// TIA Portal V20 export
FUNCTION "06 T10 LANT Output" : Void   // FC1693, LAD
TITLE = OUTPUT
{ S7_Optimized_Access := 'TRUE' }
// stored: AutoNumber false, SetENOAutomatically false
   VAR_TEMP
      Aux_real : Real;
      Aux_dint : DInt;
      Aux_uint : UInt;
      Aux_Bool : Bool;
      Aux_OS : Bool;
   END_VAR
   VAR_TEMP   // added for the SCL form of the ladder/FBD networks
      _w1 : Bool;
      _w2 : Bool;
      _w3 : Bool;
   END_VAR
BEGIN

REGION Network 1: ============= INTERLOCKS MOVING FORWARD =============
END_REGION

REGION Network 2: Interlocks Move FORWARD - Permanent Conditions
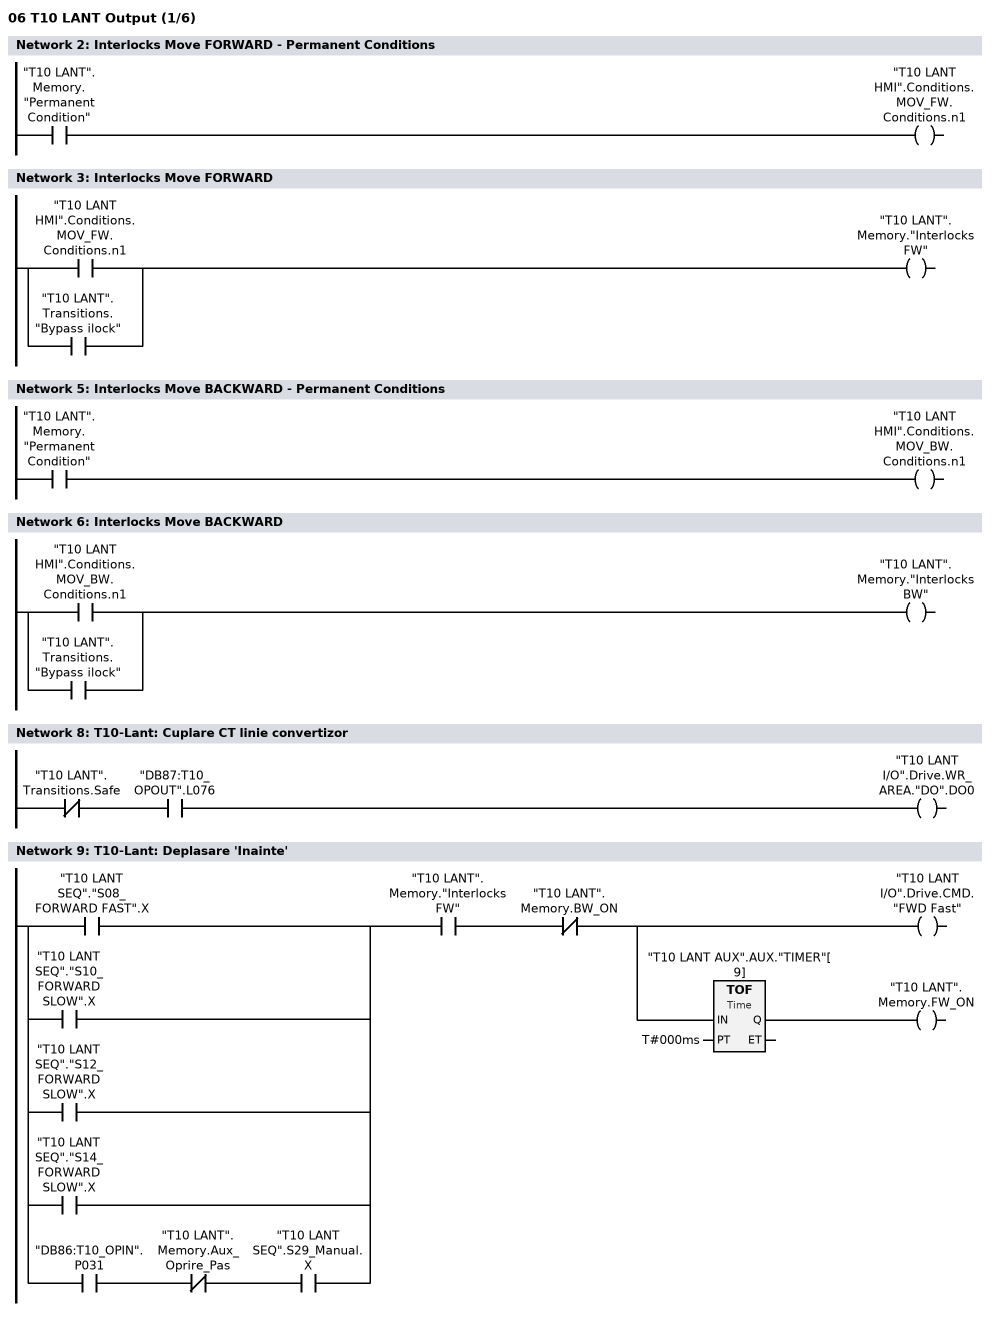
   RUNG wire#powerrail
      Contact( "T10 LANT".Memory."Permanent Condition" )
      Coil( "T10 LANT HMI".Conditions.MOV_FW.Conditions.n1 )
   END_RUNG
   // the same network as SCL:
   "T10 LANT HMI".Conditions.MOV_FW.Conditions.n1 := "T10 LANT".Memory."Permanent Condition";
END_REGION

REGION Network 3: Interlocks Move FORWARD
   RUNG wire#powerrail
      Contact( "T10 LANT HMI".Conditions.MOV_FW.Conditions.n1 )
      wire#w1
      Coil( "T10 LANT".Memory."Interlocks FW" )
   END_RUNG
   RUNG wire#powerrail
      Contact( "T10 LANT".Transitions."Bypass ilock" )
   END_RUNG wire#w1
   // the same network as SCL:
   "T10 LANT".Memory."Interlocks FW" := "T10 LANT HMI".Conditions.MOV_FW.Conditions.n1 OR "T10 LANT".Transitions."Bypass ilock";
END_REGION

REGION Network 4: ============= INTERLOCKS MOVING BACKWARD =============
END_REGION

REGION Network 5: Interlocks Move BACKWARD - Permanent Conditions
   RUNG wire#powerrail
      Contact( "T10 LANT".Memory."Permanent Condition" )
      Coil( "T10 LANT HMI".Conditions.MOV_BW.Conditions.n1 )
   END_RUNG
   // the same network as SCL:
   "T10 LANT HMI".Conditions.MOV_BW.Conditions.n1 := "T10 LANT".Memory."Permanent Condition";
END_REGION

REGION Network 6: Interlocks Move BACKWARD
   RUNG wire#powerrail
      Contact( "T10 LANT HMI".Conditions.MOV_BW.Conditions.n1 )
      wire#w1
      Coil( "T10 LANT".Memory."Interlocks BW" )
   END_RUNG
   RUNG wire#powerrail
      Contact( "T10 LANT".Transitions."Bypass ilock" )
   END_RUNG wire#w1
   // the same network as SCL:
   "T10 LANT".Memory."Interlocks BW" := "T10 LANT HMI".Conditions.MOV_BW.Conditions.n1 OR "T10 LANT".Transitions."Bypass ilock";
END_REGION

REGION Network 7: ============ COMMANDS ============
END_REGION

REGION Network 8: T10-Lant: Cuplare CT linie convertizor
   RUNG wire#powerrail
      I_Contact( "T10 LANT".Transitions.Safe )
      Contact( "DB87:T10_OPOUT".L076 )
      Coil( "T10 LANT I/O".Drive.WR_AREA."DO".DO0 )
   END_RUNG
   // the same network as SCL:
   "T10 LANT I/O".Drive.WR_AREA."DO".DO0 := NOT "T10 LANT".Transitions.Safe AND "DB87:T10_OPOUT".L076;
END_REGION

REGION Network 9: T10-Lant: Deplasare 'Inainte'
   RUNG wire#powerrail
      Contact( "T10 LANT SEQ"."S08_FORWARD FAST".X )
      wire#w1
      Contact( "T10 LANT".Memory."Interlocks FW" )
      I_Contact( "T10 LANT".Memory.BW_ON )
      wire#w2
      Coil( "T10 LANT I/O".Drive.CMD."FWD Fast" )
   END_RUNG
   RUNG wire#powerrail
      Contact( "T10 LANT SEQ"."S10_FORWARD SLOW".X )
   END_RUNG wire#w1
   RUNG wire#powerrail
      Contact( "T10 LANT SEQ"."S12_FORWARD SLOW".X )
   END_RUNG wire#w1
   RUNG wire#powerrail
      Contact( "T10 LANT SEQ"."S14_FORWARD SLOW".X )
   END_RUNG wire#w1
   RUNG wire#powerrail
      Contact( "DB86:T10_OPIN".P031 )
      I_Contact( "T10 LANT".Memory.Aux_Oprire_Pas )
      Contact( "T10 LANT SEQ".S29_Manual.X )
   END_RUNG wire#w1
   RUNG wire#w2
      { S7_Templates := "time_type := Time" } "T10 LANT AUX".AUX."TIMER"[9].TOF(pt := T#000ms, et =>)
      Coil( "T10 LANT".Memory.FW_ON )
   END_RUNG
   // the same network as SCL:
   "T10 LANT I/O".Drive.CMD."FWD Fast" := ("T10 LANT SEQ"."S08_FORWARD FAST".X OR "T10 LANT SEQ"."S10_FORWARD SLOW".X OR "T10 LANT SEQ"."S12_FORWARD SLOW".X OR "T10 LANT SEQ"."S14_FORWARD SLOW".X OR ("DB86:T10_OPIN".P031 AND NOT "T10 LANT".Memory.Aux_Oprire_Pas AND "T10 LANT SEQ".S29_Manual.X)) AND "T10 LANT".Memory."Interlocks FW" AND NOT "T10 LANT".Memory.BW_ON;
   "T10 LANT AUX".AUX."TIMER"[9].TOF(IN := "T10 LANT I/O".Drive.CMD."FWD Fast", PT := T#000ms);
   "T10 LANT".Memory.FW_ON := "T10 LANT AUX".AUX."TIMER"[9].Q;
END_REGION

REGION Network 10: T10-Lant: Deplasare 'Inapoi'
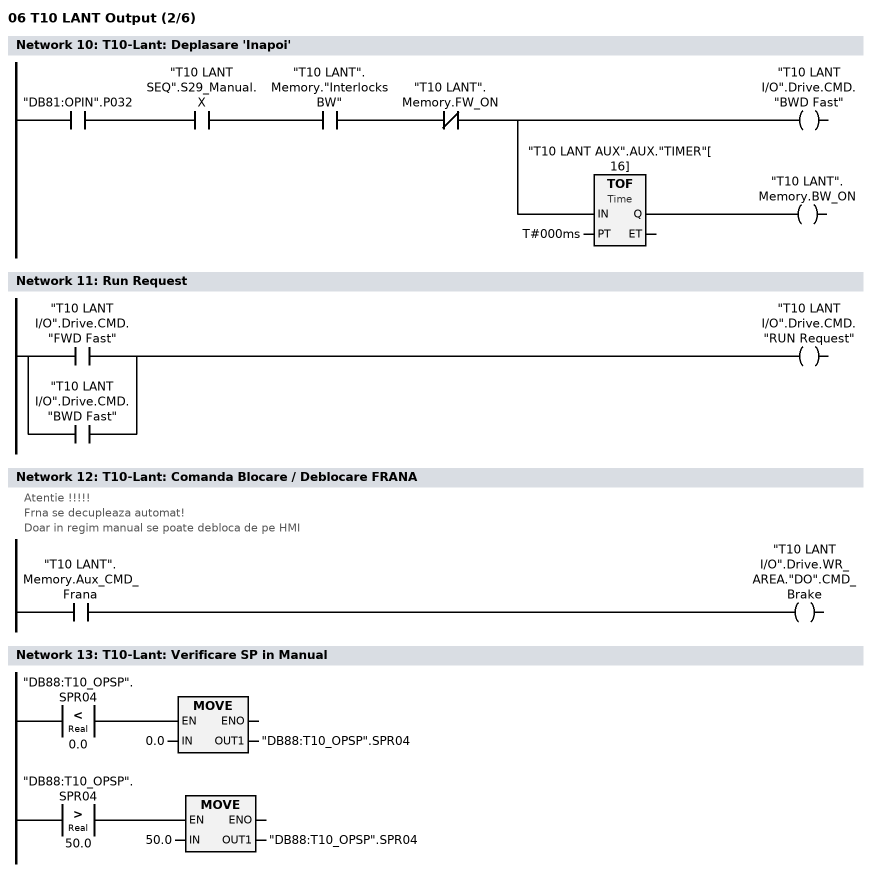
   RUNG wire#powerrail
      Contact( "DB81:OPIN".P032 )
      Contact( "T10 LANT SEQ".S29_Manual.X )
      Contact( "T10 LANT".Memory."Interlocks BW" )
      I_Contact( "T10 LANT".Memory.FW_ON )
      wire#w1
      Coil( "T10 LANT I/O".Drive.CMD."BWD Fast" )
   END_RUNG
   RUNG wire#w1
      { S7_Templates := "time_type := Time" } "T10 LANT AUX".AUX."TIMER"[16].TOF(pt := T#000ms, et =>)
      Coil( "T10 LANT".Memory.BW_ON )
   END_RUNG
   // the same network as SCL:
   "T10 LANT I/O".Drive.CMD."BWD Fast" := "DB81:OPIN".P032 AND "T10 LANT SEQ".S29_Manual.X AND "T10 LANT".Memory."Interlocks BW" AND NOT "T10 LANT".Memory.FW_ON;
   "T10 LANT AUX".AUX."TIMER"[16].TOF(IN := "T10 LANT I/O".Drive.CMD."BWD Fast", PT := T#000ms);
   "T10 LANT".Memory.BW_ON := "T10 LANT AUX".AUX."TIMER"[16].Q;
END_REGION

REGION Network 11: Run Request
   RUNG wire#powerrail
      Contact( "T10 LANT I/O".Drive.CMD."FWD Fast" )
      wire#w1
      Coil( "T10 LANT I/O".Drive.CMD."RUN Request" )
   END_RUNG
   RUNG wire#powerrail
      Contact( "T10 LANT I/O".Drive.CMD."BWD Fast" )
   END_RUNG wire#w1
   // the same network as SCL:
   "T10 LANT I/O".Drive.CMD."RUN Request" := "T10 LANT I/O".Drive.CMD."FWD Fast" OR "T10 LANT I/O".Drive.CMD."BWD Fast";
END_REGION

REGION Network 12: T10-Lant: Comanda Blocare / Deblocare FRANA
   // Atentie !!!!!
   // Frna se decupleaza automat!
   // Doar in regim manual se poate debloca de pe HMI
   RUNG wire#powerrail
      Contact( "T10 LANT".Memory.Aux_CMD_Frana )
      Coil( "T10 LANT I/O".Drive.WR_AREA."DO".CMD_Brake )
   END_RUNG
   // the same network as SCL:
   "T10 LANT I/O".Drive.WR_AREA."DO".CMD_Brake := "T10 LANT".Memory.Aux_CMD_Frana;
END_REGION

REGION Network 13: T10-Lant: Verificare SP in Manual
   RUNG wire#powerrail
      { S7_Templates := "SrcType := Real" } LT_Contact(in1 := "DB88:T10_OPSP".SPR04, in2 := 0.0)
      Move(in := 0.0, out1 => "DB88:T10_OPSP".SPR04)
   END_RUNG
   RUNG wire#powerrail
      { S7_Templates := "SrcType := Real" } GT_Contact(in1 := "DB88:T10_OPSP".SPR04, in2 := 50.0)
      Move(in := 50.0, out1 => "DB88:T10_OPSP".SPR04)
   END_RUNG
   // the same network as SCL:
   IF "DB88:T10_OPSP".SPR04 < 0.0 THEN "DB88:T10_OPSP".SPR04 := 0.0; END_IF;
   IF "DB88:T10_OPSP".SPR04 > 50.0 THEN "DB88:T10_OPSP".SPR04 := 50.0; END_IF;
END_REGION

REGION Network 14: T10-Lant: Ciclu Rapid: Viteza Referinta Incarcare
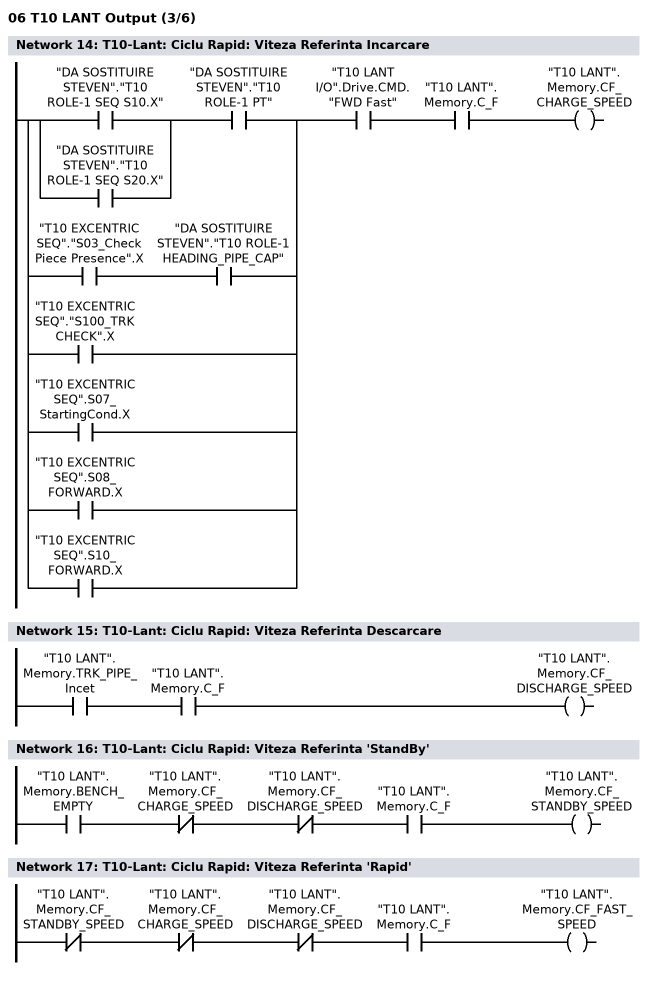
   RUNG wire#powerrail
      Contact( "DA SOSTITUIRE STEVEN"."T10 ROLE-1 SEQ S10.X" )
      wire#w1
      Contact( "DA SOSTITUIRE STEVEN"."T10 ROLE-1 PT" )
      wire#w2
      Contact( "T10 LANT I/O".Drive.CMD."FWD Fast" )
      Contact( "T10 LANT".Memory.C_F )
      Coil( "T10 LANT".Memory.CF_CHARGE_SPEED )
   END_RUNG
   RUNG wire#powerrail
      Contact( "DA SOSTITUIRE STEVEN"."T10 ROLE-1 SEQ S20.X" )
   END_RUNG wire#w1
   RUNG wire#powerrail
      Contact( "T10 EXCENTRIC SEQ"."S03_Check Piece Presence".X )
      Contact( "DA SOSTITUIRE STEVEN"."T10 ROLE-1 HEADING_PIPE_CAP" )
   END_RUNG wire#w2
   RUNG wire#powerrail
      Contact( "T10 EXCENTRIC SEQ"."S100_TRK CHECK".X )
   END_RUNG wire#w2
   RUNG wire#powerrail
      Contact( "T10 EXCENTRIC SEQ".S07_StartingCond.X )
   END_RUNG wire#w2
   RUNG wire#powerrail
      Contact( "T10 EXCENTRIC SEQ".S08_FORWARD.X )
   END_RUNG wire#w2
   RUNG wire#powerrail
      Contact( "T10 EXCENTRIC SEQ".S10_FORWARD.X )
   END_RUNG wire#w2
   // the same network as SCL:
   "T10 LANT".Memory.CF_CHARGE_SPEED := ((("DA SOSTITUIRE STEVEN"."T10 ROLE-1 SEQ S10.X" OR "DA SOSTITUIRE STEVEN"."T10 ROLE-1 SEQ S20.X") AND "DA SOSTITUIRE STEVEN"."T10 ROLE-1 PT") OR ("T10 EXCENTRIC SEQ"."S03_Check Piece Presence".X AND "DA SOSTITUIRE STEVEN"."T10 ROLE-1 HEADING_PIPE_CAP") OR "T10 EXCENTRIC SEQ"."S100_TRK CHECK".X OR "T10 EXCENTRIC SEQ".S07_StartingCond.X OR "T10 EXCENTRIC SEQ".S08_FORWARD.X OR "T10 EXCENTRIC SEQ".S10_FORWARD.X) AND "T10 LANT I/O".Drive.CMD."FWD Fast" AND "T10 LANT".Memory.C_F;
END_REGION

REGION Network 15: T10-Lant: Ciclu Rapid: Viteza Referinta Descarcare
   RUNG wire#powerrail
      Contact( "T10 LANT".Memory.TRK_PIPE_Incet )
      Contact( "T10 LANT".Memory.C_F )
      Coil( "T10 LANT".Memory.CF_DISCHARGE_SPEED )
   END_RUNG
   // the same network as SCL:
   "T10 LANT".Memory.CF_DISCHARGE_SPEED := "T10 LANT".Memory.TRK_PIPE_Incet AND "T10 LANT".Memory.C_F;
END_REGION

REGION Network 16: T10-Lant: Ciclu Rapid: Viteza Referinta 'StandBy'
   RUNG wire#powerrail
      Contact( "T10 LANT".Memory.BENCH_EMPTY )
      I_Contact( "T10 LANT".Memory.CF_CHARGE_SPEED )
      I_Contact( "T10 LANT".Memory.CF_DISCHARGE_SPEED )
      Contact( "T10 LANT".Memory.C_F )
      Coil( "T10 LANT".Memory.CF_STANDBY_SPEED )
   END_RUNG
   // the same network as SCL:
   "T10 LANT".Memory.CF_STANDBY_SPEED := "T10 LANT".Memory.BENCH_EMPTY AND NOT "T10 LANT".Memory.CF_CHARGE_SPEED AND NOT "T10 LANT".Memory.CF_DISCHARGE_SPEED AND "T10 LANT".Memory.C_F;
END_REGION

REGION Network 17: T10-Lant: Ciclu Rapid: Viteza Referinta 'Rapid'
   RUNG wire#powerrail
      I_Contact( "T10 LANT".Memory.CF_STANDBY_SPEED )
      I_Contact( "T10 LANT".Memory.CF_CHARGE_SPEED )
      I_Contact( "T10 LANT".Memory.CF_DISCHARGE_SPEED )
      Contact( "T10 LANT".Memory.C_F )
      Coil( "T10 LANT".Memory.CF_FAST_SPEED )
   END_RUNG
   // the same network as SCL:
   "T10 LANT".Memory.CF_FAST_SPEED := NOT "T10 LANT".Memory.CF_STANDBY_SPEED AND NOT "T10 LANT".Memory.CF_CHARGE_SPEED AND NOT "T10 LANT".Memory.CF_DISCHARGE_SPEED AND "T10 LANT".Memory.C_F;
END_REGION

NETWORK
TITLE = T10-Lant: Viteza Teava 'Inainte' in Mod Automat [%]
// 13.6 m/min ...... 50 Hz
// a m/min...........b Hz
// 
// b=(a*50)/13.6

      A     "T10 LANT".Memory.CF_DISCHARGE_SPEED;
      L     "PRESET POINT ACTIVE".TAB1.P93;  // DISCHARGE SPEE CYCLE
      L     1;
      /I;
      JC    _02;  // ----------------------------
      A     "T10 LANT".Memory.CF_CHARGE_SPEED;
      L     "PRESET POINT ACTIVE".TAB1.P92;  // CHARGE SPEED FAST CYCLE
      L     1;
      /I;
      JC    _02;  // ----------------------------
      A     "T10 LANT".Memory.CF_FAST_SPEED;
      L     "PRESET POINT ACTIVE".TAB1.P90;  // FAST SPEED FAST CYCLE
      L     1;
      /I;
      JC    _02;  // ----------------------------
      A     "T10 LANT".Memory.CF_STANDBY_SPEED;
      L     "PRESET POINT ACTIVE".TAB1.P91;  // STAND-BY SPEED FAST CYCLE
      L     1;
      /I;
      JC    _02;  // ----------------------------
      L     "PRESET POINT ACTIVE".TAB1.P86;  // STANDARD AUTOMATIC CYCLE
      L     1;
      /I;
_02:  NOP   0;  // ----------------------------
      ITD;
      DTR;
      T     "T10 LANT".Memory.SPEED_FW_AUTO_HZ;

      L     "T10 LANT".Memory.SPEED_FW_AUTO_HZ;
      L     50.0;
      *R;
      T     "T10 LANT".Memory.SPEED_FW_AUTO_HZ;

      L     "T10 LANT".Memory.SPEED_FW_AUTO_HZ;
      L     100.0;
      /R;
      T     "T10 LANT".Memory.SPEED_FW_AUTO_HZ;


NETWORK
TITLE = T10-Lant: Viteza Teava 'Inainte' in Mod Manual [%]
// 13.6 m/min ...... 50 Hz
// a m/min...........b Hz
// 
// b=(a*50)/13.6

      L     "PRESET POINT ACTIVE".TAB1.P87;
      L     1;
      /I;
      ITD;
      DTR;
      L     50.0;
      *R;
      L     100.0;
      /R;
      T     #Aux_real;


REGION Network 20: T10-Lant: Comenzi - Setpoint
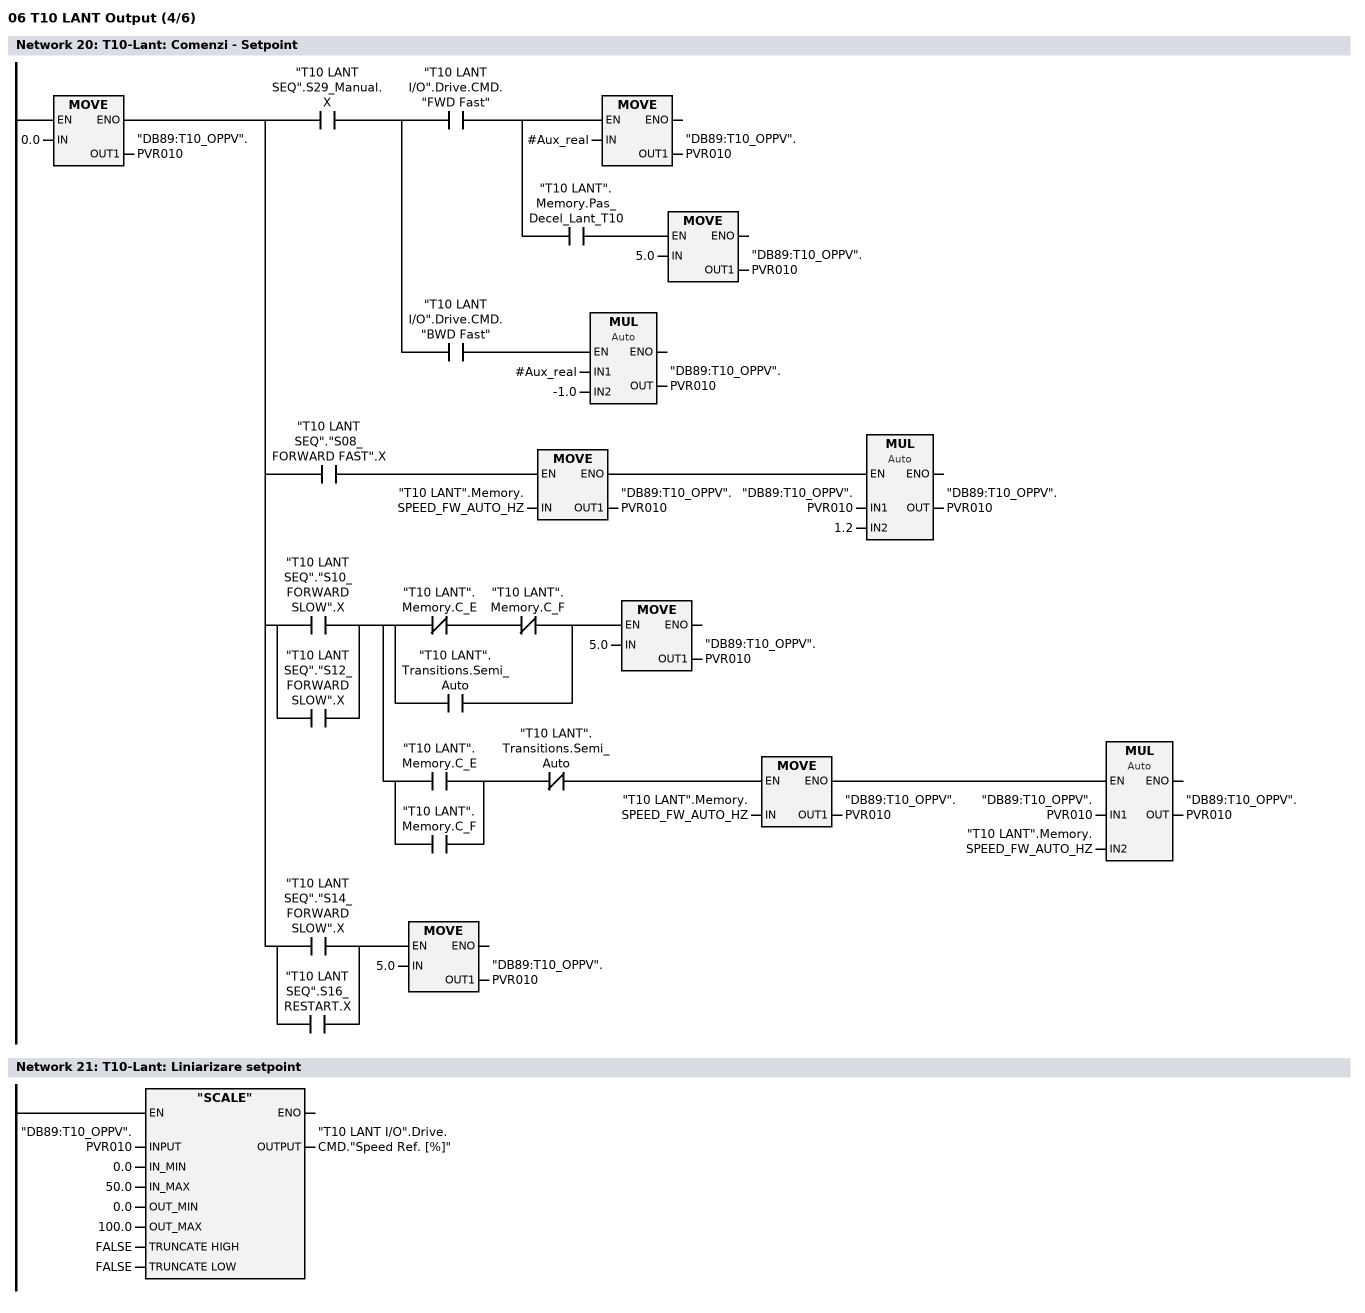
   RUNG wire#powerrail
      Move(in := 0.0, out1 => "DB89:T10_OPPV".PVR010)
      wire#w1
      Contact( "T10 LANT SEQ".S29_Manual.X )
      wire#w2
      Contact( "T10 LANT I/O".Drive.CMD."FWD Fast" )
      wire#w3
      Move(in := #Aux_real, out1 => "DB89:T10_OPPV".PVR010)
   END_RUNG
   RUNG wire#w3
      Contact( "T10 LANT".Memory.Pas_Decel_Lant_T10 )
      Move(in := 5.0, out1 => "DB89:T10_OPPV".PVR010)
   END_RUNG
   RUNG wire#w2
      Contact( "T10 LANT I/O".Drive.CMD."BWD Fast" )
      Mul(in1 := #Aux_real, in2 := -1.0, out => "DB89:T10_OPPV".PVR010)
   END_RUNG
   RUNG wire#w1
      Contact( "T10 LANT SEQ"."S08_FORWARD FAST".X )
      Move(in := "T10 LANT".Memory.SPEED_FW_AUTO_HZ, out1 => "DB89:T10_OPPV".PVR010)
      Mul(in1 := "DB89:T10_OPPV".PVR010, in2 := 1.2, out => "DB89:T10_OPPV".PVR010)
   END_RUNG
   RUNG wire#w1
      Contact( "T10 LANT SEQ"."S10_FORWARD SLOW".X )
      wire#w4
      I_Contact( "T10 LANT".Memory.C_E )
      I_Contact( "T10 LANT".Memory.C_F )
      wire#w5
      Move(in := 5.0, out1 => "DB89:T10_OPPV".PVR010)
   END_RUNG
   RUNG wire#w1
      Contact( "T10 LANT SEQ"."S12_FORWARD SLOW".X )
   END_RUNG wire#w4
   RUNG wire#w4
      Contact( "T10 LANT".Transitions.Semi_Auto )
   END_RUNG wire#w5
   RUNG wire#w4
      Contact( "T10 LANT".Memory.C_E )
      wire#w6
      I_Contact( "T10 LANT".Transitions.Semi_Auto )
      Move(in := "T10 LANT".Memory.SPEED_FW_AUTO_HZ, out1 => "DB89:T10_OPPV".PVR010)
      Mul(in1 := "DB89:T10_OPPV".PVR010, in2 := "T10 LANT".Memory.SPEED_FW_AUTO_HZ, out => "DB89:T10_OPPV".PVR010)
   END_RUNG
   RUNG wire#w4
      Contact( "T10 LANT".Memory.C_F )
   END_RUNG wire#w6
   RUNG wire#w1
      Contact( "T10 LANT SEQ"."S14_FORWARD SLOW".X )
      wire#w7
      Move(in := 5.0, out1 => "DB89:T10_OPPV".PVR010)
   END_RUNG
   RUNG wire#w1
      Contact( "T10 LANT SEQ".S16_RESTART.X )
   END_RUNG wire#w7
   // the same network as SCL:
   "DB89:T10_OPPV".PVR010 := 0.0;
   #_w1 := "T10 LANT SEQ".S29_Manual.X AND "T10 LANT I/O".Drive.CMD."FWD Fast";
   IF #_w1 THEN "DB89:T10_OPPV".PVR010 := #Aux_real; END_IF;
   IF #_w1 AND "T10 LANT".Memory.Pas_Decel_Lant_T10 THEN "DB89:T10_OPPV".PVR010 := 5.0; END_IF;
   IF "T10 LANT SEQ".S29_Manual.X AND "T10 LANT I/O".Drive.CMD."BWD Fast" THEN
       "DB89:T10_OPPV".PVR010 := #Aux_real * (-1.0);
   END_IF;
   IF "T10 LANT SEQ"."S08_FORWARD FAST".X THEN
       "DB89:T10_OPPV".PVR010 := "T10 LANT".Memory.SPEED_FW_AUTO_HZ;
       "DB89:T10_OPPV".PVR010 := "DB89:T10_OPPV".PVR010 * 1.2;
   END_IF;
   #_w2 := "T10 LANT SEQ"."S10_FORWARD SLOW".X OR "T10 LANT SEQ"."S12_FORWARD SLOW".X;
   IF #_w2 AND ((NOT "T10 LANT".Memory.C_E AND NOT "T10 LANT".Memory.C_F) OR "T10 LANT".Transitions.Semi_Auto) THEN
       "DB89:T10_OPPV".PVR010 := 5.0;
   END_IF;
   IF #_w2 AND ("T10 LANT".Memory.C_E OR "T10 LANT".Memory.C_F) AND NOT "T10 LANT".Transitions.Semi_Auto THEN
       "DB89:T10_OPPV".PVR010 := "T10 LANT".Memory.SPEED_FW_AUTO_HZ;
       "DB89:T10_OPPV".PVR010 := "DB89:T10_OPPV".PVR010 * "T10 LANT".Memory.SPEED_FW_AUTO_HZ;
   END_IF;
   IF "T10 LANT SEQ"."S14_FORWARD SLOW".X OR "T10 LANT SEQ".S16_RESTART.X THEN
       "DB89:T10_OPPV".PVR010 := 5.0;
   END_IF;
END_REGION

REGION Network 21: T10-Lant: Liniarizare setpoint
   RUNG wire#powerrail
      "SCALE"(INPUT := "DB89:T10_OPPV".PVR010, IN_MIN := 0.0, IN_MAX := 50.0, OUT_MIN := 0.0, OUT_MAX := 100.0, "TRUNCATE HIGH" := FALSE, "TRUNCATE LOW" := FALSE, OUTPUT => "T10 LANT I/O".Drive.CMD."Speed Ref. [%]")
   END_RUNG
   // the same network as SCL:
   "SCALE"(INPUT := "DB89:T10_OPPV".PVR010,
           IN_MIN := 0.0,
           IN_MAX := 50.0,
           OUT_MIN := 0.0,
           OUT_MAX := 100.0,
           "TRUNCATE HIGH" := FALSE,
           "TRUNCATE LOW" := FALSE,
           OUTPUT => "T10 LANT I/O".Drive.CMD."Speed Ref. [%]");
END_REGION

REGION Network 22: T10-Lant: Functie convertizor
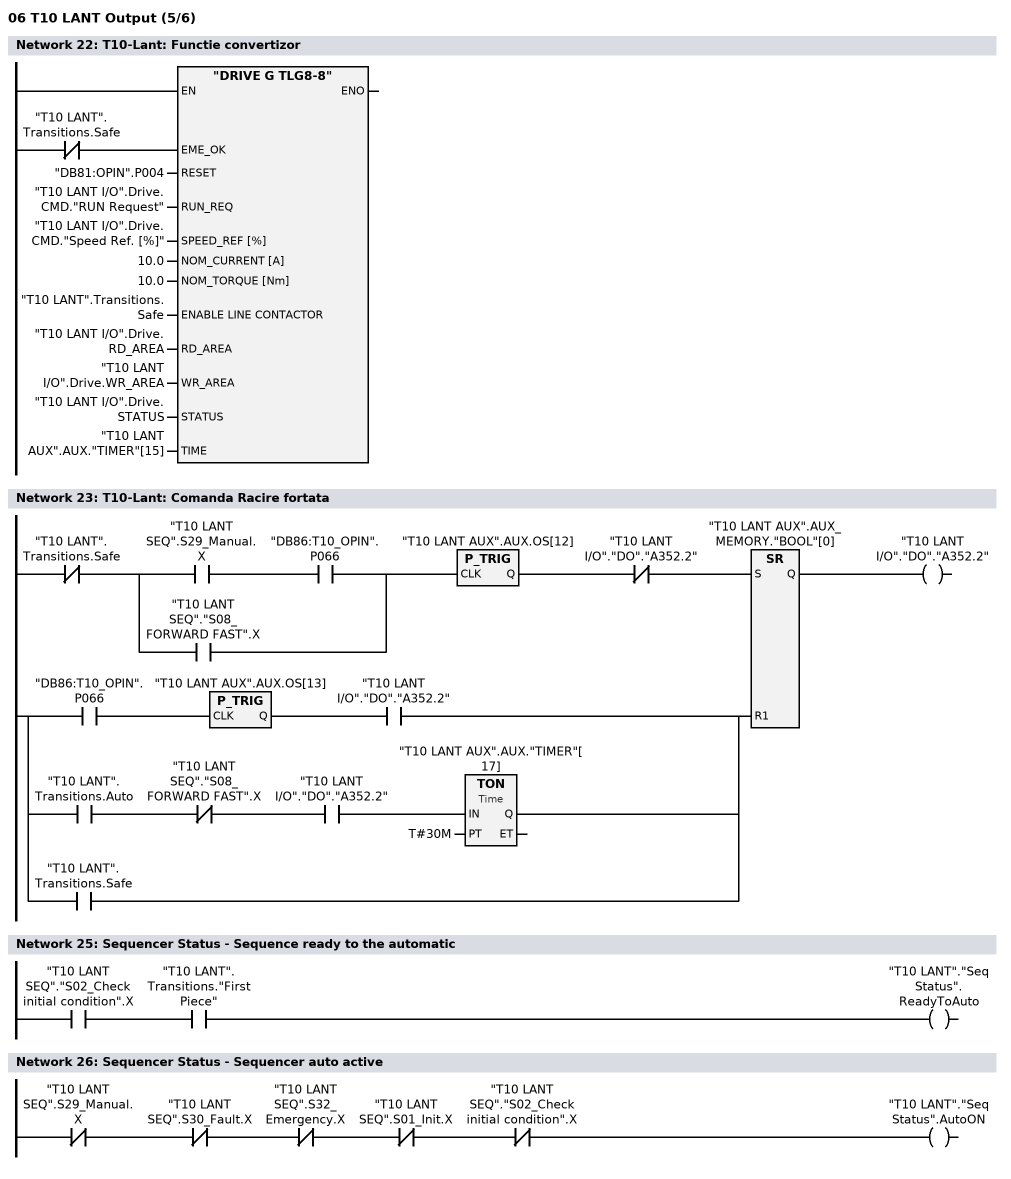
   RUNG wire#powerrail
      "DRIVE G TLG8-8"(EME_OK := wire#w1, RESET := "DB81:OPIN".P004, RUN_REQ := "T10 LANT I/O".Drive.CMD."RUN Request", "SPEED_REF [%]" := "T10 LANT I/O".Drive.CMD."Speed Ref. [%]", "NOM_CURRENT [A]" := 10.0, "NOM_TORQUE [Nm]" := 10.0, "ENABLE LINE CONTACTOR" := "T10 LANT".Transitions.Safe, RD_AREA := "T10 LANT I/O".Drive.RD_AREA, WR_AREA := "T10 LANT I/O".Drive.WR_AREA, STATUS := "T10 LANT I/O".Drive.STATUS, "TIME" := "T10 LANT AUX".AUX."TIMER"[15])
   END_RUNG
   RUNG wire#powerrail
      I_Contact( "T10 LANT".Transitions.Safe )
   END_RUNG wire#w1
   // the same network as SCL:
   "DRIVE G TLG8-8"(EME_OK := NOT "T10 LANT".Transitions.Safe,
                    RESET := "DB81:OPIN".P004,
                    RUN_REQ := "T10 LANT I/O".Drive.CMD."RUN Request",
                    "SPEED_REF [%]" := "T10 LANT I/O".Drive.CMD."Speed Ref. [%]",
                    "NOM_CURRENT [A]" := 10.0,
                    "NOM_TORQUE [Nm]" := 10.0,
                    "ENABLE LINE CONTACTOR" := "T10 LANT".Transitions.Safe,
                    RD_AREA := "T10 LANT I/O".Drive.RD_AREA,
                    WR_AREA := "T10 LANT I/O".Drive.WR_AREA,
                    STATUS := "T10 LANT I/O".Drive.STATUS,
                    "TIME" := "T10 LANT AUX".AUX."TIMER"[15]);
END_REGION

REGION Network 23: T10-Lant: Comanda Racire fortata
   RUNG wire#powerrail
      I_Contact( "T10 LANT".Transitions.Safe )
      wire#w1
      Contact( "T10 LANT SEQ".S29_Manual.X )
      Contact( "DB86:T10_OPIN".P066 )
      wire#w2
      P_Trig( "T10 LANT AUX".AUX.OS[12] )
      I_Contact( "T10 LANT I/O"."DO"."A352.2" )
      S_SR(operand := "T10 LANT AUX".AUX_MEMORY."BOOL"[0], r1 := wire#w3)
      Coil( "T10 LANT I/O"."DO"."A352.2" )
   END_RUNG
   RUNG wire#w1
      Contact( "T10 LANT SEQ"."S08_FORWARD FAST".X )
   END_RUNG wire#w2
   RUNG wire#powerrail
      Contact( "DB86:T10_OPIN".P066 )
      P_Trig( "T10 LANT AUX".AUX.OS[13] )
      Contact( "T10 LANT I/O"."DO"."A352.2" )
   END_RUNG wire#w3
   RUNG wire#powerrail
      Contact( "T10 LANT".Transitions.Auto )
      I_Contact( "T10 LANT SEQ"."S08_FORWARD FAST".X )
      Contact( "T10 LANT I/O"."DO"."A352.2" )
      { S7_Templates := "time_type := Time" } "T10 LANT AUX".AUX."TIMER"[17].TON(pt := T#30M, et =>)
   END_RUNG wire#w3
   RUNG wire#powerrail
      Contact( "T10 LANT".Transitions.Safe )
   END_RUNG wire#w3
   // the same network as SCL:
   #_w1 := NOT "T10 LANT".Transitions.Safe AND (("T10 LANT SEQ".S29_Manual.X AND "DB86:T10_OPIN".P066) OR "T10 LANT SEQ"."S08_FORWARD FAST".X);
   #_w2 := #_w1 AND NOT "T10 LANT AUX".AUX.OS[12];   // rising edge
   "T10 LANT AUX".AUX.OS[12] := #_w1;
   #_w3 := "DB86:T10_OPIN".P066 AND NOT "T10 LANT AUX".AUX.OS[13];   // rising edge
   "T10 LANT AUX".AUX.OS[13] := "DB86:T10_OPIN".P066;
   "T10 LANT AUX".AUX."TIMER"[17].TON(IN := "T10 LANT".Transitions.Auto AND NOT "T10 LANT SEQ"."S08_FORWARD FAST".X AND "T10 LANT I/O"."DO"."A352.2",
                           PT := T#30M);
   IF #_w2 AND NOT "T10 LANT I/O"."DO"."A352.2" THEN
       "T10 LANT AUX".AUX_MEMORY."BOOL"[0] := TRUE;   // SR flip-flop
   END_IF;
   IF (#_w3 AND "T10 LANT I/O"."DO"."A352.2") OR "T10 LANT AUX".AUX."TIMER"[17].Q OR "T10 LANT".Transitions.Safe THEN
       "T10 LANT AUX".AUX_MEMORY."BOOL"[0] := FALSE;
   END_IF;
   "T10 LANT I/O"."DO"."A352.2" := "T10 LANT AUX".AUX_MEMORY."BOOL"[0];
END_REGION

REGION Network 24: ================== SEQUENCER STATUS ==================
END_REGION

REGION Network 25: Sequencer Status - Sequence ready to the automatic
   RUNG wire#powerrail
      Contact( "T10 LANT SEQ"."S02_Check initial condition".X )
      Contact( "T10 LANT".Transitions."First Piece" )
      Coil( "T10 LANT"."Seq Status".ReadyToAuto )
   END_RUNG
   // the same network as SCL:
   "T10 LANT"."Seq Status".ReadyToAuto := "T10 LANT SEQ"."S02_Check initial condition".X AND "T10 LANT".Transitions."First Piece";
END_REGION

REGION Network 26: Sequencer Status - Sequencer auto active
   RUNG wire#powerrail
      I_Contact( "T10 LANT SEQ".S29_Manual.X )
      I_Contact( "T10 LANT SEQ".S30_Fault.X )
      I_Contact( "T10 LANT SEQ".S32_Emergency.X )
      I_Contact( "T10 LANT SEQ".S01_Init.X )
      I_Contact( "T10 LANT SEQ"."S02_Check initial condition".X )
      Coil( "T10 LANT"."Seq Status".AutoON )
   END_RUNG
   // the same network as SCL:
   "T10 LANT"."Seq Status".AutoON := NOT "T10 LANT SEQ".S29_Manual.X AND NOT "T10 LANT SEQ".S30_Fault.X AND NOT "T10 LANT SEQ".S32_Emergency.X AND NOT "T10 LANT SEQ".S01_Init.X AND NOT "T10 LANT SEQ"."S02_Check initial condition".X;
END_REGION

REGION Network 27: Sequencer Status - Sequencer wait piece
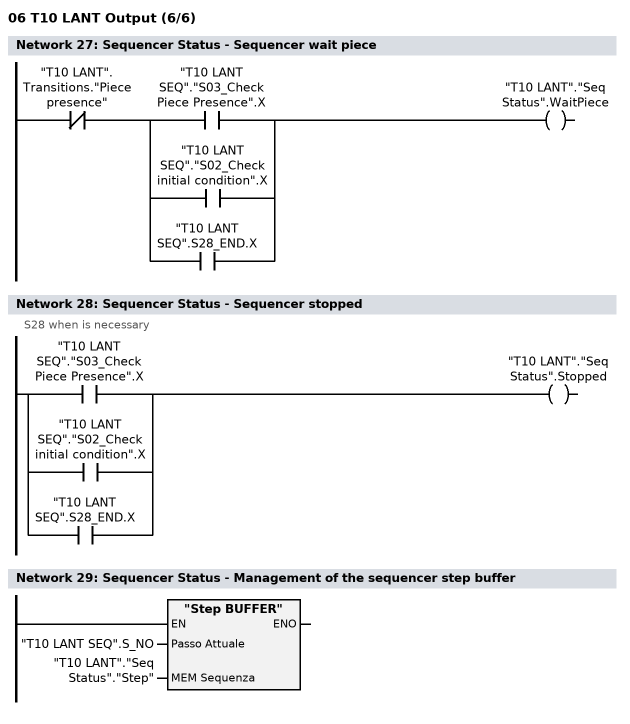
   RUNG wire#powerrail
      I_Contact( "T10 LANT".Transitions."Piece presence" )
      wire#w1
      Contact( "T10 LANT SEQ"."S03_Check Piece Presence".X )
      wire#w2
      Coil( "T10 LANT"."Seq Status".WaitPiece )
   END_RUNG
   RUNG wire#w1
      Contact( "T10 LANT SEQ"."S02_Check initial condition".X )
   END_RUNG wire#w2
   RUNG wire#w1
      Contact( "T10 LANT SEQ".S28_END.X )
   END_RUNG wire#w2
   // the same network as SCL:
   "T10 LANT"."Seq Status".WaitPiece := NOT "T10 LANT".Transitions."Piece presence" AND ("T10 LANT SEQ"."S03_Check Piece Presence".X OR "T10 LANT SEQ"."S02_Check initial condition".X OR "T10 LANT SEQ".S28_END.X);
END_REGION

REGION Network 28: Sequencer Status - Sequencer stopped
   // S28 when is necessary
   RUNG wire#powerrail
      Contact( "T10 LANT SEQ"."S03_Check Piece Presence".X )
      wire#w1
      Coil( "T10 LANT"."Seq Status".Stopped )
   END_RUNG
   RUNG wire#powerrail
      Contact( "T10 LANT SEQ"."S02_Check initial condition".X )
   END_RUNG wire#w1
   RUNG wire#powerrail
      Contact( "T10 LANT SEQ".S28_END.X )
   END_RUNG wire#w1
   // the same network as SCL:
   "T10 LANT"."Seq Status".Stopped := "T10 LANT SEQ"."S03_Check Piece Presence".X OR "T10 LANT SEQ"."S02_Check initial condition".X OR "T10 LANT SEQ".S28_END.X;
END_REGION

REGION Network 29: Sequencer Status - Management of the sequencer step buffer
   RUNG wire#powerrail
      "Step BUFFER"("Passo Attuale" := "T10 LANT SEQ".S_NO, "MEM Sequenza" := "T10 LANT"."Seq Status"."Step")
   END_RUNG
   // the same network as SCL:
   "Step BUFFER"("Passo Attuale" := "T10 LANT SEQ".S_NO, "MEM Sequenza" := "T10 LANT"."Seq Status"."Step");
END_REGION
END_FUNCTION
